(* IEC 61131-3 sources: AXOpen/src/showcase/app/src/components.drives/Documentation/TypesStructuresAndEnums, 3 files *)

(* ---- AxoDrive_Control_Example.st ---- *)
NAMESPACE AXOpen.Components.Drives
    {S7.extern=ReadWrite}
    {#ix-attr:[Container(Layout.Tabs)]}
    CLASS PUBLIC AxoDrive_Control_Example
        VAR PUBLIC
            {#ix-set:AttributeName = "<#DriveControlWord#>"}
            DriveControlWord : WORD;
            {#ix-set:AttributeName = "<#CommandPosition#>"}
            CommandPosition : DINT;
            {#ix-set:AttributeName = "<#CommandVelocity#>"}
            CommandVelocity : DINT;
            {#ix-set:AttributeName = "<#CommandAcceleration#>"}
            CommandAcceleration : DINT;
            {#ix-set:AttributeName = "<#CommandDecceleration#>"}
            CommandDecceleration : DINT;
            {#ix-set:AttributeName = "<#CommandTorque#>"}
            CommandTorque : INT;
            {#ix-set:AttributeName = "<#CommandJerk#>"}
            CommandJerk : DINT;
        END_VAR
    END_CLASS
END_NAMESPACE

(* ---- AxoDrive_HWIDs_Example.st ---- *)
NAMESPACE AXOpen.Components.Drives
   {S7.extern=ReadWrite}
	CLASS AxoDrive_HWIDs_Example
      VAR PUBLIC
         {#ix-set:AttributeName = "<#Hardware ID Device#>"}
         HW_Device            : UINT;
         {#ix-set:AttributeName = "<#Hardware ID 'Outputs' module#>"}
         HW_Outputs           : UINT;
         {#ix-set:AttributeName = "<#Hardware ID 'Inputs' module#>"}
         HW_Inputs            : UINT;
         {#ix-set:AttributeName = "<#Hardware ID 'S_0_0134_0_0__Servodrive_profile__Control_word' submodule#>"}
         HW_S_0_0134_0_0      : UINT;
         {#ix-set:AttributeName = "<#Hardware ID 'S_0_0282_0_0__Drive_controlled_positioning__Command_value' submodule#>"}
         HW_S_0_0282_0_0      : UINT;
         {#ix-set:AttributeName = "<#Hardware ID 'S_0_0259_0_0__Positioning_profile__Profile_velocity' submodule#>"}
         HW_S_0_0259_0_0      : UINT;
         {#ix-set:AttributeName = "<#Hardware ID 'S_0_0260_0_0__Positioning_profile__Acceleration' submodule#>"}
         HW_S_0_0260_0_0      : UINT;
         {#ix-set:AttributeName = "<#Hardware ID 'S_0_0359_0_0__Positioning_profile__Deceleration' submodule#>"}
         HW_S_0_0359_0_0      : UINT;
         {#ix-set:AttributeName = "<#Hardware ID 'S_0_0080_0_0__Torque_force_command_value' submodule#>"}
         HW_S_0_0080_0_0      : UINT;
         {#ix-set:AttributeName = "<#Hardware ID 'S_0_0193_0_0__Positioning_jerk' submodule#>"}
         HW_S_0_0193_0_0      : UINT;
         {#ix-set:AttributeName = "<#Hardware ID 'S_0_0135_0_0__Servodrive_profile__Status_word' submodule#>"}
         HW_S_0_0135_0_0      : UINT;
         {#ix-set:AttributeName = "<#Hardware ID 'S_0_0386_0_0__Position_controller__Position_actual_value' submodule#>"}
         HW_S_0_0386_0_0      : UINT;
         {#ix-set:AttributeName = "<#Hardware ID 'S_0_0535_0_0__Velocity_controller__Velocity_actual_value' submodule#>"}
         HW_S_0_0535_0_0      : UINT;
         {#ix-set:AttributeName = "<#Hardware ID 'S_0_0390_0_0__Diagnostic_message__Manufacturer_status_register' submodule#>"}
         HW_S_0_0390_0_0      : UINT;
         {#ix-set:AttributeName = "<#Hardware ID 'S_0_0084_0_0__Torque_force_feedback_value' submodule#>"}
         HW_S_0_0084_0_0      : UINT;
      END_VAR
   END_CLASS
END_NAMESPACE

(* ---- AxoDriveAxisRefExample.st ---- *)
USING AXOpen.Core;
USING AXOpen.Messaging.Static;
USING AXOpen.Messaging;
USING AXOpen.Core;
USING AXOpen.Components.Abstractions;
USING AXOpen.Components.Abstractions.Drives;

NAMESPACE AXOpen.Components.Drives
    {S7.extern=ReadWrite}
    CLASS AxoDriveAxisReferenceExample IMPLEMENTS AXOpen.Components.Abstractions.Drives.IAxoAxisReference
        VAR PUBLIC // HWin
            {#ix-attr:[Container(Layout.Stack)]}
            {#ix-attr:[ComponentDetails("HW inputs")]}
            {#ix-attr:[ReadOnly()]}
            Inputs  :   AxoDrive_Status_Example;
        END_VAR
        VAR PUBLIC // HWout
            {#ix-attr:[Container(Layout.Stack)]}
            {#ix-attr:[ComponentDetails("HW outputs")]}
            {#ix-attr:[ReadOnly()]}
            Outputs  :   AxoDrive_Control_Example;
        END_VAR
        VAR PUBLIC // HWIDs
            {#ix-attr:[Container(Layout.Stack)]}
            {#ix-attr:[ComponentDetails("HWids")]}
            {#ix-attr:[ReadOnly()]}
            HWIDs  :   AxoDrive_HWIDs_Example;
        END_VAR
        VAR PUBLIC // Data
            {#ix-attr:[Container(Layout.Stack)]}
            {#ix-attr:[ComponentDetails("Data")]}
            {#ix-attr:[ReadOnly()]}
            Data            :   AxoDrive_Data_Example;
        END_VAR
        VAR PUBLIC
            Config          :   AXOpen.Components.Drives.AxoDrive_Config;
            Status          :   AXOpen.Components.Drives.AxoDrive_Status;
        END_VAR
    END_CLASS
END_NAMESPACE
